// TIA Portal V16 export
// export: Created 2024-12-03T15:41:41.3475694Z, ExportSetting WithDefaults, DisplayName Totally Integrated Automation Portal, DisplayVersion V16 Update 6, DisplayName TIA Portal Version Control Interface, DisplayVersion V16 Update 2, DisplayName TIA Portal Openness, DisplayVersion V16 Update 6, DisplayName TIA Portal Teamcenter Gateway, DisplayVersion V16, DisplayName SINAMICS Startdrive Advanced, DisplayVersion V16 Update 5, DisplayName SINAMICS Startdrive G130, G150, S120, S150, SINAMICS MV, S210, DisplayVersion V16 Update 5, DisplayName SINAMICS Startdrive G110M, G120, G120C, G120D, G120P, G115D, DisplayVersion V16 Update 5, DisplayName STEP 7 Professional, DisplayVersion V16 Update 6, DisplayName STEP 7 Safety, DisplayVersion V16, DisplayName WinCC Advanced / Unified PC, DisplayVersion V16 Update 6
FUNCTION_BLOCK "Virtual_Encoder_FB"   // FB45, SCL
{ S7_Optimized_Access := 'TRUE' }
VERSION : 0.1
// stored: AutoNumber true, IsIECCheckEnabled false, IsRetainMemResEnabled false, MemoryReserve 100, SetENOAutomatically false, UDAEnableTagReadback false
   VAR_INPUT
      I_RelativeReferenceSpeed_Perc : Real;   // %
      I_AbsoluteSpeedOnReferecne_m_min : Real;   // m/min
      I_CurrentRelativeSpeed_Perc : Real;   // %
   END_VAR
   VAR_OUTPUT
      O_Delta_mm : Real;
   END_VAR
   VAR_IN_OUT
      IO_VirtualEncoder : "VirtualEncoder_UDT";
   END_VAR
   VAR
      cycleTime : "ScanTimer_FB";
   END_VAR
   VAR_TEMP
      T_Gain : Real;
      T_CurrentSpeed_mm_ms : Real;
      T_Distance_mm : Real;
   END_VAR
BEGIN
   REGION Calculate absolute speed on 100% relative speed

       #T_Gain := #I_AbsoluteSpeedOnReferecne_m_min / #I_RelativeReferenceSpeed_Perc; // scale to 1% m/min
       #T_Gain := (#T_Gain * 1000.0) / 60.0; // scale to mm/s
       #T_Gain := #T_Gain / 1000.0; // scale to mm/ms

   END_REGION

   REGION Calculate abosulte speed

       #T_CurrentSpeed_mm_ms := #T_Gain * #I_CurrentRelativeSpeed_Perc;

   END_REGION

   REGION Call scantimer

       #cycleTime();

   END_REGION

   REGION Determine absolute distance

       #T_Distance_mm := #T_CurrentSpeed_mm_ms * DINT_TO_REAL(#cycleTime.O_ScanTime);
       #O_Delta_mm := #T_Distance_mm;

       #IO_VirtualEncoder.Distance_mm := #O_Delta_mm;
       #IO_VirtualEncoder.Speed_mm_ms := #T_CurrentSpeed_mm_ms;

   END_REGION
END_FUNCTION_BLOCK
